(* CODESYS project StringBuilder32_Itfs.library
   Description: Interfaces for StringBuilder32
   Version: 0.5.0.0
   Title: StringBuilder Interfaces32
   Author: John te Bokkel
   DocFormat: reStructuredText
   Placeholder: StringBuilder Interfaces
   LanguageModelAttribute: qualified-access-only
   Company: PowerCore Engineering
   DefaultNamespace: PSBItfs

Project tree, tasks and I/O mapping:
  StringBuilder_Itfs/
    Enums/
      data type ERROR
    GlobalConstants/
    Interfaces/
      interface IStringBuilder: p_length, Append, Reset, p_CharBufferPtr
    Structs/
    Types/
*)

// StringBuilder_Itfs/Enums/ERROR
{attribute 'qualified_only'}
TYPE ERROR : (NO_ERROR, TIME_OUT); END_TYPE

// StringBuilder_Itfs/Interfaces/IStringBuilder
INTERFACE IStringBuilder EXTENDS __SYSTEM.IQueryInterface

PROPERTY p_length : UDINT
GET
END_GET
END_PROPERTY

/// Append ``sVal`` to the string
METHOD Append : INT
VAR_INPUT
	sVal : STRING(255);
END_VAR
END_METHOD

/// Clears the string and resets append position
METHOD Reset : BOOL
VAR_INPUT
END_VAR
END_METHOD

PROPERTY p_CharBufferPtr : POINTER TO BYTE
GET
END_GET
END_PROPERTY

END_INTERFACE
